Omron CX-Programmer project NuevoProyecto (CX-Programmer 9.61)

# PLC NuevoPLC1: CQM1 CPU41

## Program NuevoPrograma1 (no task)
Local symbols
KMD 100.05 BOOL  ; Contactor marcha derecha
KMI 100.02 BOOL  ; Contactor marcha izquierda
LA 100.13 BOOL  ; Lámpara de avería
LF 100.14 BOOL  ; Lámpara de funcionamiento
PM 0.02 BOOL  ; Pulsador de marcha
PMD 0.05 BOOL  ; Pulsador marcha derecha
PMI 0.02 BOOL
PP 0.15 BOOL  ; Pulsador de paro
RT 0.13 BOOL  ; Contacto relé térmico

### Section Sección1

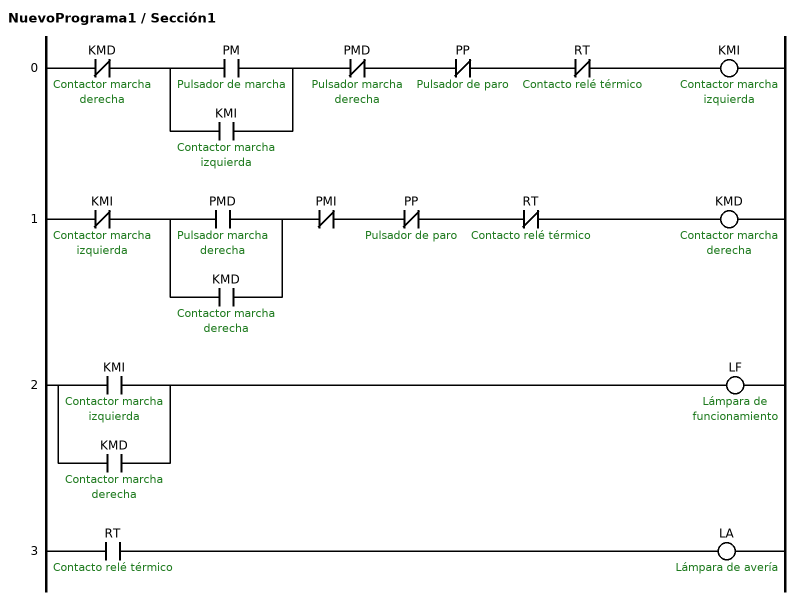
; rung 0
LDNOT KMD  ; Contactor marcha derecha
LD PM  ; Pulsador de marcha
OR KMI  ; Contactor marcha izquierda
ANDLD
ANDNOT PMD  ; Pulsador marcha derecha
ANDNOT PP  ; Pulsador de paro
ANDNOT RT  ; Contacto relé térmico
OUT KMI  ; Contactor marcha izquierda
; rung 1
LDNOT KMI  ; Contactor marcha izquierda
LD PMD  ; Pulsador marcha derecha
OR KMD  ; Contactor marcha derecha
ANDLD
ANDNOT PMI
ANDNOT PP  ; Pulsador de paro
ANDNOT RT  ; Contacto relé térmico
OUT KMD  ; Contactor marcha derecha
; rung 2
LD KMI  ; Contactor marcha izquierda
OR KMD  ; Contactor marcha derecha
OUT LF  ; Lámpara de funcionamiento
; rung 3
LD RT  ; Contacto relé térmico
OUT LA  ; Lámpara de avería

### Section END
; rung 0
END(01)